// TIA Portal V19 export
ORGANIZATION_BLOCK "TestCallEnv"   // OB10000, FBD, ProgramCycle
TITLE = "Main Program Sweep (Cycle)"
{ S7_Optimized_Access := 'TRUE' }
// #@AutoGenerated
// stored: SetENOAutomatically false
   VAR_INPUT
      Initial_Call : Bool;   // Initial call of this OB
      Remanence : Bool;   // =True, if remanent data are available
   END_VAR
BEGIN

REGION Network 1: : Call LPythagorean - AppTest LPythagoreanTestCase
   // #@AutoGenerated
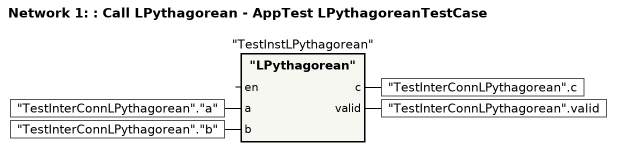
   "TestInstLPythagorean"("a" := "TestInterConnLPythagorean"."a",   // "LPythagorean"
                          "b" := "TestInterConnLPythagorean"."b",
                          c => "TestInterConnLPythagorean".c,
                          valid => "TestInterConnLPythagorean".valid);
END_REGION
END_ORGANIZATION_BLOCK
